PROGRAM p_InitVariable
VAR
END_VAR

END_PROGRAM

(* stored: Version 1.1.0.1, ProductVersion 3.1.4020.6
   POU p_InitVariable: Id {85af2f83-c6cf-4831-908b-8edd5e0fc377}, SpecialFunc None *)
